# EPICS autosave request: tests/testfiles/cfg/SF_Movers_PV.req
$(SYS):X_SP
$(SYS):Y_SP
$(SYS):ROT_X_SP
$(SYS):ROT_Y_SP
$(SYS):ROT_Z_SP
